TYPE REQUEST_ :
STRUCT
	Command			:UINT;		// Value according to the command table
	Data			:ARRAY[0..18] OF UINT := [0];
END_STRUCT
END_TYPE

(* stored: Version 1.1.0.1
   DUT REQUEST_: Id {3aa5f61e-7445-40e0-af08-832e24592a20} *)
